# EPICS substitutions: CsHeaterApp/Db/Watlow_PM_Loop_PID.substitutions
file Watlow_PM_Loop_PID.template
{
pattern	{  s, ta,      ss, mod, ch}
        { '', SE,  Watlow,   1,  1}
}
